// Mitsubishi GX Works2 project: servo_motor_2   PLC: Q02/Q02H

PROGRAM MAIN
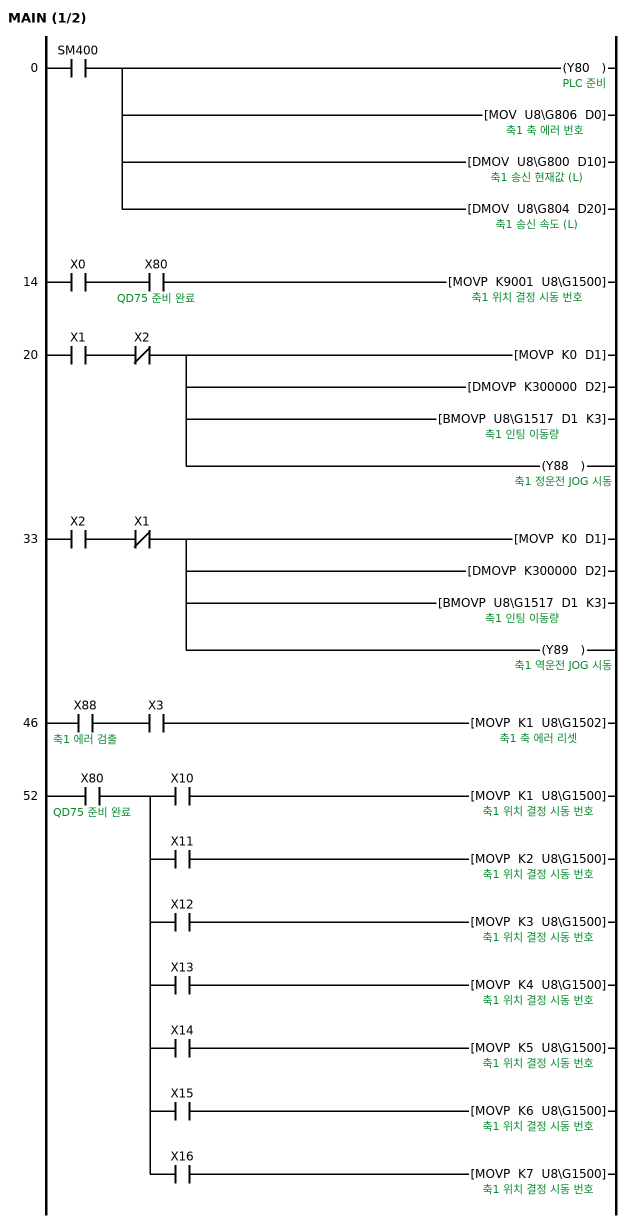
0     LD      SM400
      OUT     Y80  ; PLC 준비
      MOV     U8\G806 D0  ; 축1 축 에러 번호
      DMOV    U8\G800 D10  ; 축1 송신 현재값 (L)
      DMOV    U8\G804 D20  ; 축1 송신 속도 (L)
14    LD      X0
      AND     X80  ; QD75 준비 완료
      MOVP    K9001 U8\G1500  ; 축1 위치 결정 시동 번호
20    LD      X1
      ANI     X2
      MOVP    K0 D1
      DMOVP   K300000 D2
      BMOVP   U8\G1517 D1 K3  ; 축1 인팅 이동량
      OUT     Y88  ; 축1 정운전 JOG 시동
33    LD      X2
      ANI     X1
      MOVP    K0 D1
      DMOVP   K300000 D2
      BMOVP   U8\G1517 D1 K3
      OUT     Y89  ; 축1 역운전 JOG 시동
46    LD      X88  ; 축1 에러 검출
      AND     X3
      MOVP    K1 U8\G1502  ; 축1 축 에러 리셋
52    LD      X80  ; QD75 준비 완료
      MPS
      AND     X10
      MOVP    K1 U8\G1500
      MRD
      AND     X11
      MOVP    K2 U8\G1500
      MRD
      AND     X12
      MOVP    K3 U8\G1500
      MRD
      AND     X13
      MOVP    K4 U8\G1500
      MRD
      AND     X14
      MOVP    K5 U8\G1500
      MRD
      AND     X15
      MOVP    K6 U8\G1500
      MPP
      AND     X16
      MOVP    K7 U8\G1500
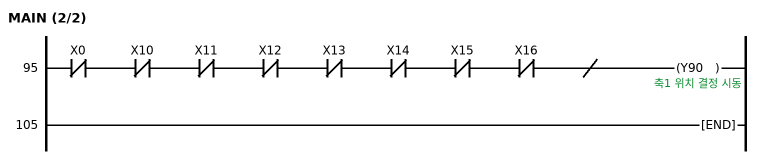
95    LDI     X0
      ANI     X10
      ANI     X11
      ANI     X12
      ANI     X13
      ANI     X14
      ANI     X15
      ANI     X16
      INV
      OUT     Y90  ; 축1 위치 결정 시동
105   END
END_PROGRAM

PROGRAM no_intel
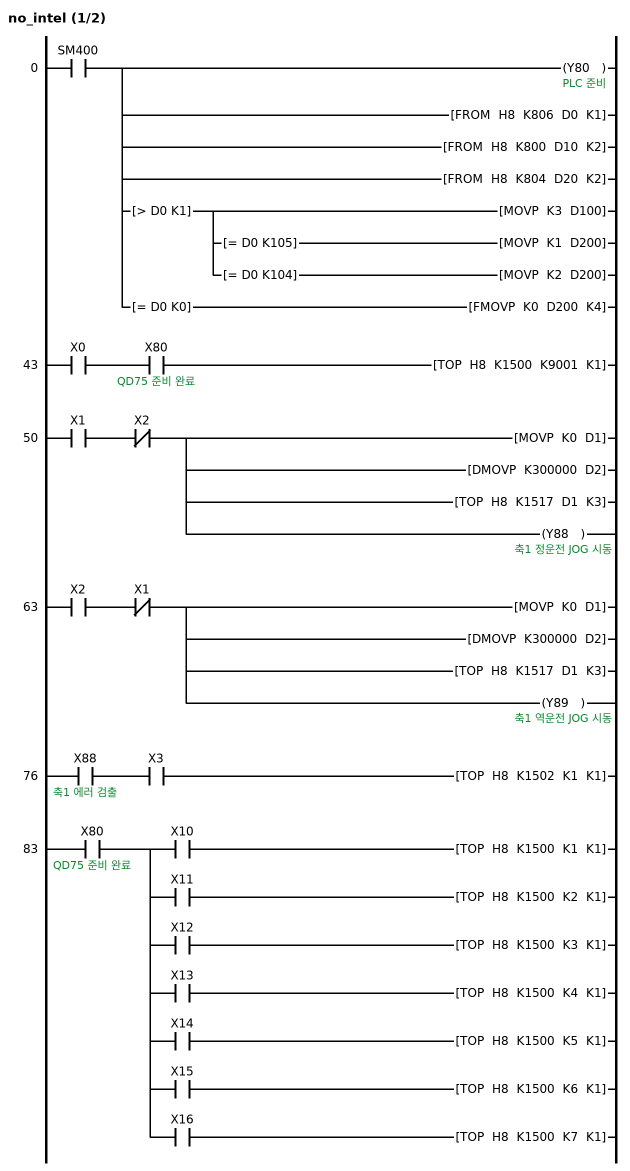
0     LD      SM400
      OUT     Y80  ; PLC 준비
      FROM    H8 K806 D0 K1
      FROM    H8 K800 D10 K2
      FROM    H8 K804 D20 K2
      MPS
      AND>    D0 K1
      MOVP    K3 D100
      MPS
      AND=    D0 K105
      MOVP    K1 D200
      MPP
      AND=    D0 K104
      MOVP    K2 D200
      MPP
      AND=    D0 K0
      FMOVP   K0 D200 K4
43    LD      X0
      AND     X80  ; QD75 준비 완료
      TOP     H8 K1500 K9001 K1
50    LD      X1
      ANI     X2
      MOVP    K0 D1
      DMOVP   K300000 D2
      TOP     H8 K1517 D1 K3
      OUT     Y88  ; 축1 정운전 JOG 시동
63    LD      X2
      ANI     X1
      MOVP    K0 D1
      DMOVP   K300000 D2
      TOP     H8 K1517 D1 K3
      OUT     Y89  ; 축1 역운전 JOG 시동
76    LD      X88  ; 축1 에러 검출
      AND     X3
      TOP     H8 K1502 K1 K1
83    LD      X80  ; QD75 준비 완료
      MPS
      AND     X10
      TOP     H8 K1500 K1 K1
      MRD
      AND     X11
      TOP     H8 K1500 K2 K1
      MRD
      AND     X12
      TOP     H8 K1500 K3 K1
      MRD
      AND     X13
      TOP     H8 K1500 K4 K1
      MRD
      AND     X14
      TOP     H8 K1500 K5 K1
      MRD
      AND     X15
      TOP     H8 K1500 K6 K1
      MPP
      AND     X16
      TOP     H8 K1500 K7 K1
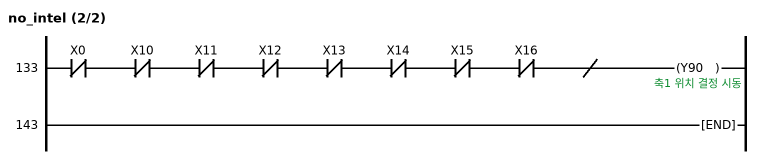
133   LDI     X0
      ANI     X10
      ANI     X11
      ANI     X12
      ANI     X13
      ANI     X14
      ANI     X15
      ANI     X16
      INV
      OUT     Y90  ; 축1 위치 결정 시동
143   END
END_PROGRAM

PROGRAM HMI
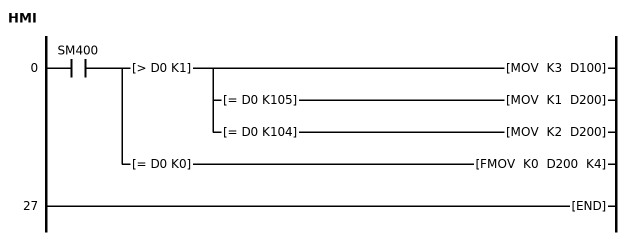
0     LD      SM400
      MPS
      AND>    D0 K1
      MOV     K3 D100
      MPS
      AND=    D0 K105
      MOV     K1 D200
      MPP
      AND=    D0 K104
      MOV     K2 D200
      MPP
      AND=    D0 K0
      FMOV    K0 D200 K4
27    END
END_PROGRAM

// device comments not shown above
X81  ; 동기용 플래그
X84  ; 축1 M 코드 ON
X85  ; 축2 M 코드 ON
X89  ; 축2 에러 검출
X8C  ; 축1 BUSY
X8D  ; 축2 BUSY
X90  ; 축1 시동 완료
X91  ; 축2 시동 완료
X94  ; 축1 위치 결정 완료
X95  ; 축2 위치 결정 완료
Y84  ; 축1 축 정지
Y85  ; 축2 축 정지
Y8A  ; 축2 정운전 JOG 시동
Y8B  ; 축2 역운전 JOG 시동
Y91  ; 축2 위치 결정 시동
Y94  ; 축1 실행 금지 플래그
Y95  ; 축2 실행 금지 플래그
